{attribute addProperty BoxType "EJ9576-0000-0019"}
{attribute addProperty Id "Terminal_OvertemperatureAT %I*BOOL811I2T_errorAT %I*BOOL812I2T_warningAT %I*BOOL813OvervoltageAT %I*BOOL814UndervoltageAT %I*BOOL815Chopper_onAT %I*BOOL816Input_cycle_counterAT %I*BYTE8115DC_link_voltageAT %I*UDINT32417Resistor_currentAT %I*DINT32419Duty_cylceAT %I*USINT8120I2T_load_factorAT %I*USINT8121"}
{attribute addProperty CRC "1782415764"}
{attribute addProperty SizeInBites "136"}
{attribute addProperty SizeInBytes "17"}
TYPE BCT_Inputs_6A3D8194 :
STRUCT
	{attribute addProperty Name "Terminal_Overtemperature"}
	Terminal_Overtemperature AT %I* : BOOL;
	{attribute addProperty Name "I2T_error"}
	I2T_error AT %I* : BOOL;
	{attribute addProperty Name "I2T_warning"}
	I2T_warning AT %I* : BOOL;
	{attribute addProperty Name "Overvoltage"}
	Overvoltage AT %I* : BOOL;
	{attribute addProperty Name "Undervoltage"}
	Undervoltage AT %I* : BOOL;
	{attribute addProperty Name "Chopper_on"}
	Chopper_on AT %I* : BOOL;
	{attribute addProperty Name "Input_cycle_counter"}
	Input_cycle_counter AT %I* : BYTE;
	{attribute addProperty Name "DC_link_voltage"}
	DC_link_voltage AT %I* : UDINT;
	{attribute addProperty Name "Resistor_current"}
	Resistor_current AT %I* : DINT;
	{attribute addProperty Name "Duty_cylce"}
	Duty_cylce AT %I* : USINT;
	{attribute addProperty Name "I2T_load_factor"}
	I2T_load_factor AT %I* : USINT;
END_STRUCT
END_TYPE

(* stored: Version 1.2.0.0, ProductVersion 3.1.4024.9
   DUT BCT_Inputs_6A3D8194: Id {8e6a1508-cb67-4d7a-80e2-2ca8cd7b43f6} *)
